RoboDK station: 机器人绘图工作站.rdk

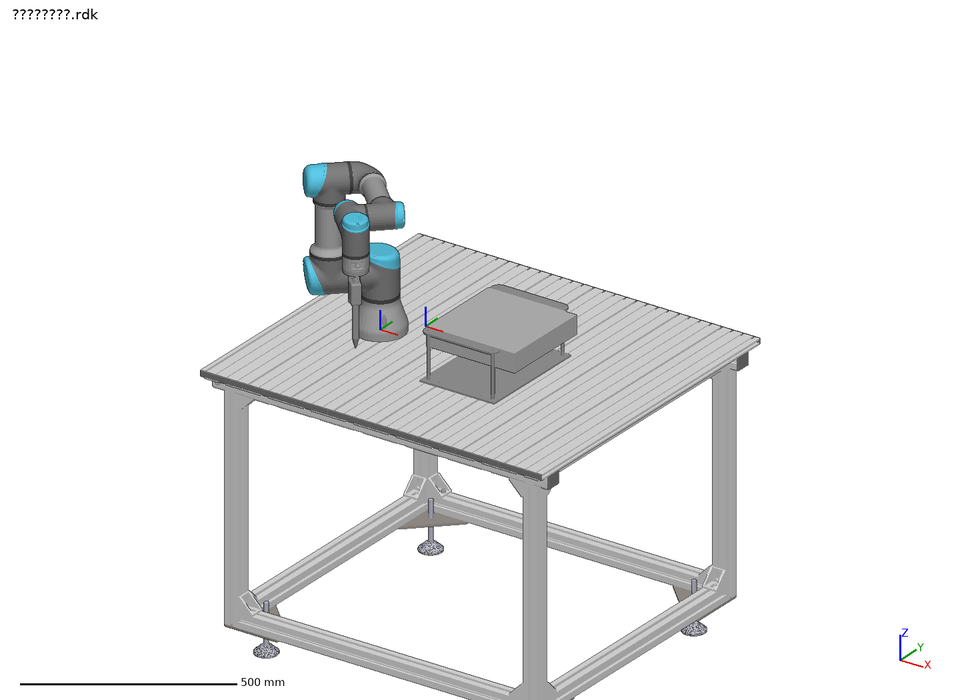
[picture v0: the station drawn from its stored meshes, robots at their saved joint values, targets as dots, program paths as lines]
Station 机器人绘图工作站. Poses are relative to the parent item; angles as X-Y-Z fixed-axis rotations.
  - object  at (0, 0, 0) mm, size 3 x 3 x 1 mm, geometry from .sld
  - object  at (0, 0, 0) mm, size 960 x 880 x 736.1 mm, geometry from .step
  - frame 绘图坐标系 at (200, -176.36, 13.37) mm
    - object  at (0.98, -0.26, 0) mm, size 250 x 250 x 50 mm, geometry from .sld
    - object  at (0.98, -0.26, 0) mm, size 203 x 115.1 x 51 mm, geometry from .sld
  - frame UR3 Base at (0, -72, -93) mm
    - robot UR3: 6 axes, payload 3 kg, reach 500 mm, repeatability 0.1 mm, weight 11 kg
        modified DH rows (alpha deg, a mm, theta deg, d mm): 0, 0, 0, 151.9; 90, 0, 180, 0; 0, 243.65, 0, 0; 0, 213, 0, 110.4; -90, 0, 0, 83.4; 90, 0, 180, 82.4
        joint limits [-360, -360, -360, -360, -360, -360] to [360, 360, 360, 360, 360, 360]; home [0, -90, -90, 0, 90, 0]; saved at [-45, -90, -90, -90, 90, 0]
      - tool , TCP at (0, 0, 182.9) mm, size 61 x 61 x 208 mm
  - object  at (200, -200, 10) mm, size 210.1 x 310.1 x 130 mm, geometry from .step
  - Python program simulate (listed below)

--- Python program simulate ---
from robolink import *      # 加载robolink模块
from robodk import *        # 加载robodk模块

import sys                  # 加载sys模块
import os                   # 加载os
import json

RDK = Robolink()            # 定义RoboDK工作站

path_stationfile = RDK.getParam('PATH_OPENSTATION')     # 获取当前工作站的路径
sys.path.append(os.path.abspath(path_stationfile))      # 将当前工作站的路径添加到系统路径中
# from b import *

# 定义工作站中的对象
robot = RDK.Item('UR3')            # 定义机器人对象
write_frame = RDK.Item('绘图坐标系')              # 定义写字坐标系：write_frame
write_tool = RDK.Item('书写工具')                    # 定义写字工具
pixel = RDK.Item('像素点')                        # 定义写字像素点
image_template = RDK.Item('模板')                 # 定义画板的模板
image = RDK.Item('画板')                          # 预定义工作站的画板

######## 定义函数 ###########

# 定义函数：将二维空间中的点转化为三维空间中的点（4*4矩阵）
def point2D_2_pose(point, tangent):
    return transl(point.x, point.y, 0)*rotz(tangent.angle())

# s=0，笔从不接触纸面到接触纸面
def point2D_2_pose0(point, tangent):
    return transl(point.x, point.y, )*rotz(tangent.angle())

# s=1，接触保持纸面
def point2D_2_pose1(point, tangent):
    return transl(point.x, point.y, )*rotz(tangent.angle())

# s=2，从接触纸面到离开纸面
def point2D_2_pose2(point, tangent):
    return transl(point.x, point.y, )*rotz(tangent.angle())

def write_robot(list, item_frame, item_tool, robot, bias):
    APPROACH = 34                                             # 定义常量APPROACH为100
    home_joints = [-45,-90,-90,-90,90,0]                                # 定义机器人的起始位置

    robot.setPoseFrame(item_frame)                              # 定义机器人的工件坐标系
    robot.setPoseTool(item_tool)                                # 定义机器人的工具坐标系
    robot.MoveJ(home_joints)                                    # 机器人移动到起始位置

    orient_frame2tool = roty(pi)

    for p in list:
        # p=[i*200/1024 for i in p]
        p[0]=p[0]*100/1024+80
        p[1]=p[1]*100/1024+40-bias
        if p[2]==0 or p[2]==2:
            target0 = transl(p[0], p[1], 0)*orient_frame2tool         # 将p_0转化为机器人目标点target_0(4*4矩阵)
            target0_app = target0*transl(0,0,-APPROACH-10)             # 定义目标点：target0_app
            robot.MoveL(target0_app)
        elif p[2]==1:
            target0 = transl(p[0], p[1], 0)*orient_frame2tool         # 将p_0转化为机器人目标点target_0(4*4矩阵)
            target0_app = target0*transl(0,0,-APPROACH)             # 定义目标点：target0_app
            robot.MoveL(target0_app)

    robot.MoveL(home_joints)

######## 机器人写字主程序 #########
# s = input('请输入汉字：')
# for c in range(len(s)):
    # a = pen_track(s[c])
    # a = [j for i in a for j in i]
s = '清'
json_path = os.path.join(path_stationfile,'characters_tracks.json')
with open(json_path,'r') as js:
    track = json.load(js)
a = track[s]
write_robot(a, write_frame, write_tool, robot,60)
s1 = '华'
a1 = track[s1]
write_robot(a1, write_frame, write_tool, robot,-60)
